INTERFACE I_OP_MODE_PAUSE_VISU EXTENDS I_GENERAL_OBJECT

METHOD M_ResetModeSelection : BOOL
VAR_INPUT
END_VAR
END_METHOD

PROPERTY P_BreakPressureDetSelected : BOOL
GET
END_GET
END_PROPERTY

PROPERTY P_EnduranceRunSelected : BOOL
GET
END_GET
END_PROPERTY

PROPERTY P_HandSelected : BOOL
GET
END_GET
END_PROPERTY

PROPERTY P_JogCounterCyl1_Active : BOOL
GET
END_GET
END_PROPERTY

PROPERTY P_JogCounterCyl2_Active : BOOL
GET
END_GET
END_PROPERTY

PROPERTY P_JogCounterCyl3_Active : BOOL
GET
END_GET
END_PROPERTY

PROPERTY P_JogCounterCyl4_Active : BOOL
GET
END_GET
END_PROPERTY

PROPERTY P_JogSelected : BOOL
GET
END_GET
END_PROPERTY

PROPERTY P_LeakTest1Selected : BOOL
GET
END_GET
END_PROPERTY

PROPERTY P_LeakTest2Selected : BOOL
GET
END_GET
END_PROPERTY

END_INTERFACE

(* stored: Version 1.1.0.1, ProductVersion 3.1.4024.12
   Itf I_OP_MODE_PAUSE_VISU: Id {98a1ed61-d86f-4e46-a6b6-7efb36e2fece}
   Method M_ResetModeSelection: Id {63a384db-3a1c-43ac-aeaa-eeeeec911782}
   Property P_BreakPressureDetSelected: Id {fbbc00c5-68ed-46a0-96b2-161fd5786c7c}
   Get Get: Id {ac688b97-2473-4c1b-9390-96f45d3b97c2}
   Property P_EnduranceRunSelected: Id {c7b6db4b-e9fb-4194-853b-f5e5941fe5d4}
   Get Get: Id {b45c6d21-c314-4e21-b97d-9695bd10e24e}
   Property P_HandSelected: Id {5eb67c90-4ce5-4a06-8b96-47eb9ca2fb55}
   Get Get: Id {fb2c83d9-08a9-4f89-a25f-058519a8f55d}
   Property P_JogCounterCyl1_Active: Id {b52c4b42-6d21-4b2d-aad4-b7e37f0b286f}
   Get Get: Id {f4cf070f-5755-49c7-b326-ab93d4d39c2b}
   Property P_JogCounterCyl2_Active: Id {a805c4e3-b72c-442e-bc0e-4d41093c5054}
   Get Get: Id {75c13b91-f592-4cb5-a4e6-6375f039099a}
   Property P_JogCounterCyl3_Active: Id {57462241-0504-4aff-b997-20201994a3cd}
   Get Get: Id {fb79bdcf-59e1-4ec5-b20e-f06b47209cca}
   Property P_JogCounterCyl4_Active: Id {0c3e8bb5-da4c-426a-a2df-bff19e5050b0}
   Get Get: Id {41d688c5-40d4-45fa-9dda-6b8af2bc42e9}
   Property P_JogSelected: Id {04637374-4e0e-41f1-aadf-e92d05001f89}
   Get Get: Id {e7a897e6-3cac-4a05-ae84-fcbbca5f4d3c}
   Property P_LeakTest1Selected: Id {6fe90742-f44a-4a57-85e1-e290a60aa0be}
   Get Get: Id {fb741230-1cd3-4451-9cd3-00203901e657}
   Property P_LeakTest2Selected: Id {f369598e-4229-4a10-887b-9fd48c88a926}
   Get Get: Id {36ed6580-8804-49ba-8e91-472b1dbe519a} *)
